{attribute 'GeneratedUsingTerminal: AT2050-0500-0023'}
{attribute addProperty BoxType "AT2050-0500-0023"}
{attribute addProperty Id "A_0090_AT2050_5501_0019_AT2050_5501AT2050_01D6DEDF80"}
{attribute addProperty CRC "544029625"}
{attribute addProperty Size "80"}
TYPE A_0054_AT2050_0500_0023_206D3BB9 EXTENDS AT2050_86175B41 :
STRUCT
	{attribute addProperty Name "A_0090_AT2050_5501_0019_AT2050_5501"}
	A_0090_AT2050_5501_0019_AT2050_5501 : AT2050_01D6DEDF;
END_STRUCT
END_TYPE

(* stored: Version 1.2.0.0, ProductVersion 3.1.4024.9
   DUT A_0054_AT2050_0500_0023_206D3BB9: Id {4c50c86a-22ee-4dd4-9498-2d7914276bcd} *)
